INTERFACE ITF_DeurSensor

PROPERTY DeurSensorStatus : BOOL
GET
END_GET
END_PROPERTY

END_INTERFACE

(* stored: Version 1.1.0.1
   Itf ITF_DeurSensor: Id {2f67539b-6e64-4102-bff7-e5dfcc03fad9}
   Folder Properties: Id {56e6a988-36ed-447f-bc4b-fca118618317}
   Property DeurSensorStatus: Id {081ff636-afa5-472e-8b5e-99ca006d15cc}
   Get Get: Id {513d4a95-7511-45d6-8f4c-55e88c67636f} *)
